// Mitsubishi GX Works2 project: 240430_timechart02_outoff   PLC: Q03UDV

PROGRAM MAIN
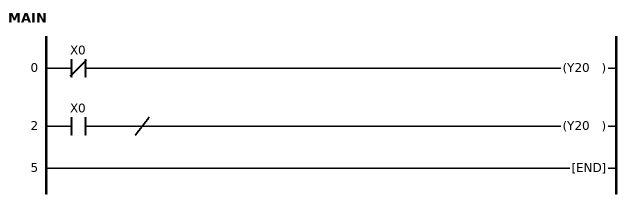
0     LDI     X0
      OUT     Y20
2     LD      X0
      INV
      OUT     Y20
5     END
END_PROGRAM
